// TIA Portal V20 export
FUNCTION_BLOCK "Clamp"   // FB431, LAD
{ S7_Optimized_Access := 'TRUE' }
// stored: AutoNumber false, MemoryReserve 100, SetENOAutomatically false
   VAR_INPUT
      Req_arms_move_to_workPos : Bool;
      Req_arms_move_to_basePos : Bool;
      BasePos1 : Bool;
      WorkPos1 : Bool;
      BasePos2 : Bool;
      WorkPos2 : Bool;
      Palette_on_station : Bool;
      Arms_in_pos : Bool;
      Hydraulic_unit_rdy : Bool;
   END_VAR
   VAR_OUTPUT
      MoveToWorkPos : Bool;
      MoveToBasePos : Bool;
   END_VAR
   VAR
      Alarm_Clamp_Not_Close_Properly { S7_SetPoint := 'True'} : TON_TIME;
      Alarm_Clamp_Not_Open_Properly { S7_SetPoint := 'True'} : TON_TIME;
   END_VAR
BEGIN

REGION Network 1: Open Clamps
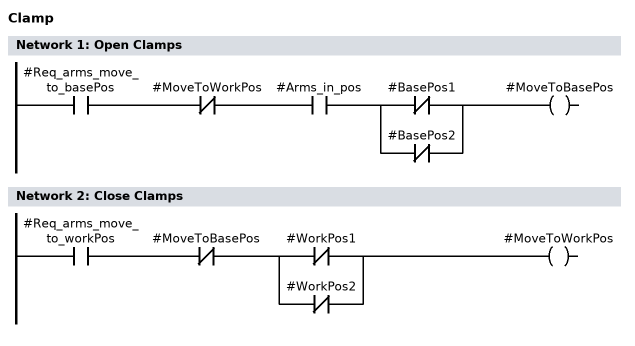
   RUNG wire#powerrail
      Contact( #Req_arms_move_to_basePos )
      I_Contact( #MoveToWorkPos )
      Contact( #Arms_in_pos )
      wire#w1
      I_Contact( #BasePos1 )
      wire#w2
      Coil( #MoveToBasePos )
   END_RUNG
   RUNG wire#w1
      I_Contact( #BasePos2 )
   END_RUNG wire#w2
   // the same network as SCL:
   #MoveToBasePos := #Req_arms_move_to_basePos AND NOT #MoveToWorkPos AND #Arms_in_pos AND (NOT #BasePos1 OR NOT #BasePos2);
END_REGION

REGION Network 2: Close Clamps
   RUNG wire#powerrail
      Contact( #Req_arms_move_to_workPos )
      I_Contact( #MoveToBasePos )
      wire#w1
      I_Contact( #WorkPos1 )
      wire#w2
      Coil( #MoveToWorkPos )
   END_RUNG
   RUNG wire#w1
      I_Contact( #WorkPos2 )
   END_RUNG wire#w2
   // the same network as SCL:
   #MoveToWorkPos := #Req_arms_move_to_workPos AND NOT #MoveToBasePos AND (NOT #WorkPos1 OR NOT #WorkPos2);
END_REGION

REGION Network 3 (SCL): Alarm Clamps not in position
   #Alarm_Clamp_Not_Close_Properly.TON(IN:=#MoveToWorkPos = 1 AND (#WorkPos1 = 0 OR #WorkPos2 = 0),
                                       PT:=T#3s);
   #Alarm_Clamp_Not_Open_Properly.TON(IN:=#MoveToBasePos = 1 AND (#BasePos1 = 0 OR #BasePos2 = 0) ,
                                       PT:=T#3s);
END_REGION
END_FUNCTION_BLOCK
